Staubli VAL3: start.pgx

program start()
begin
  userPage()
  cls()

  // feedback task will run every 32 ms (approx. 31 HZ)
  //nFbkPeriod=0.032
  nFbkPeriod=0.05
  // motion task will run every 12 ms (approx. 83 Hz)
  nMotionPeriod=0.012

  nDeg2Rad = 3.14159265359 / 180.0

  sFbkTaskName="publisher"

  // initialise TCP/IP parameters
  //call initParams()

  // create feedback (state and status) task to send data to industrial_robot)client
  taskCreateSync sFbkTaskName,nFbkPeriod,bFbkOverrun,jStateStreamer()

end
